FUNCTION_BLOCK FB_System_Fenster_Logik
VAR_IN_OUT
	Steuerung	: ST_System_Fenster_Steuerung;
	Zustand		: ST_System_Fenster_Zustand;
END_VAR
VAR_INPUT
	Parameter	: ST_System_Fenster_Parameter;
END_VAR
VAR_OUTPUT
END_VAR
VAR
END_VAR

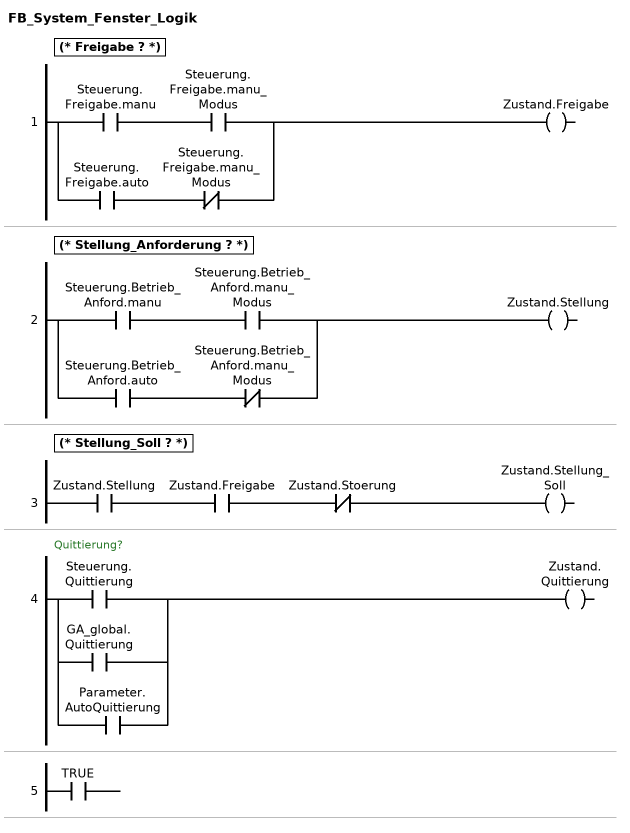
// NETWORK 1
// label: (* Freigabe ? *)
Zustand.Freigabe := Steuerung.Freigabe.manu AND Steuerung.Freigabe.manu_Modus OR Steuerung.Freigabe.auto AND NOT Steuerung.Freigabe.manu_Modus;

// NETWORK 2
// label: (* Stellung_Anforderung ? *)
Zustand.Stellung := Steuerung.Betrieb_Anford.manu AND Steuerung.Betrieb_Anford.manu_Modus OR Steuerung.Betrieb_Anford.auto AND NOT Steuerung.Betrieb_Anford.manu_Modus;

// NETWORK 3
// label: (* Stellung_Soll ? *)
Zustand.Stellung_Soll := Zustand.Stellung AND Zustand.Freigabe AND NOT Zustand.Stoerung;

// NETWORK 4
// Quittierung?
Zustand.Quittierung := Steuerung.Quittierung OR GA_global.Quittierung OR Parameter.AutoQuittierung;

// NETWORK 5

END_FUNCTION_BLOCK

(* stored: Version 1.1.0.1, ProductVersion 3.1.4024.9
   POU FB_System_Fenster_Logik: Id {6bfc897c-baf4-41e9-8b4d-eeebf98cd1c9}, SpecialFunc None *)
